(* LS Electric XG5000 project: BasicPLC *)
(* PLC LSPLC *)

PROGRAM NewProgram (* task: 스캔 프로그램 *)
VAR
    in1 : BOOL;
    inq1 : INT := 10000;
    inq1s : BOOL;
    movein : INT := 22;
    moveout : INT;
    outq1 : REAL;
    outq2 : REAL;
    outq3 : INT;
    q21 : REAL := 5;
    q22 : REAL := 3;
END_VAR

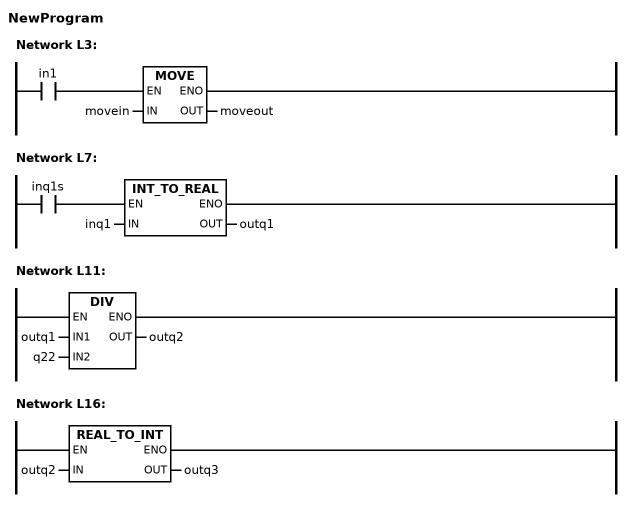
(* Rung L3 *)
IF in1 THEN moveout := movein; END_IF;
(* Rung L7 *)
IF inq1s THEN outq1 := INT_TO_REAL(inq1); END_IF;
(* Rung L11 *)
outq2 := outq1 / q22;
(* Rung L16 *)
outq3 := REAL_TO_INT(outq2);
END_PROGRAM